// TIA Portal V17 export
// export: Created 2025-06-20T11:06:35.1143958Z, ExportSetting WithDefaults, DisplayName Totally Integrated Automation Portal, DisplayVersion V17 Update 8, DisplayName TIA Portal Openness, DisplayVersion V17 Update 8, DisplayName TIA Portal Version Control Interface, DisplayVersion V17, DisplayName SINAMICS Startdrive Advanced, DisplayVersion V17 SP2, DisplayName SINAMICS Startdrive G110M, G120, G120C, G120D, G120P, G115D, DisplayVersion V17 SP2, DisplayName SINAMICS Startdrive G130, G150, S120, S150, SINAMICS MV, S210, DisplayVersion V17 SP2, DisplayName STEP 7 Professional, DisplayVersion V17 Update 8, DisplayName SINUMERIK ONE STEP 7 Toolbox, DisplayVersion V17 Update 12, DisplayName SINUMERIK ONE PLC Basic Program Plus, DisplayVersion V17 Update 12, DisplayName SINUMERIK 840D sl STEP 7 Toolbox, DisplayVersion V17 Update 12, DisplayName STEP 7 Safety, DisplayVersion V17 Update 6, DisplayName WinCC Advanced, DisplayVersion V17 Update 8
DATA_BLOCK "DB1251_PART_CYCLE_UNIT_2"   // DB1251
{ S7_Optimized_Access := 'FALSE'; DB_Accessible_From_OPC_UA := 'FALSE' }
AUTHOR : ETXETAR
VERSION : 1.0
// stored: AutoNumber false, DBAccessibleFromOPCUA false, DBAccessibleFromWebserver true, IsOnlyStoredInLoadMemory false, IsWriteProtectedInAS false
   VAR RETAIN
      SEQUENCE : "SEQUENCE";
      CYCLE_UNIT_02_STATION_0 : Bool;   // CYCLE UNIT 02 STATION 0 START REQUEST
      CYCLE_UNIT_02_STATION_1 : Bool;   // CYCLE UNIT 02 STATION 1 START REQUEST
      CYCLE_UNIT_02_STATION_2 : Bool;   // CYCLE UNIT 02 STATION 2 START REQUEST
      CYCLE_UNIT_02_STATION_3 : Bool;   // CYCLE UNIT 02 STATION 3 START REQUEST
      CYCLE_UNIT_02_STATION_4 : Bool;   // CYCLE UNIT 02 STATION 4 START REQUEST
      UNIT_02_CALIBRATION_STATION_2 : Bool;   // UNIT 02 STATION 2 CALIBRATION CYCLE REQUEST
      UNIT_02_CALIBRATION_STATION_3 : Bool;   // UNIT 02 STATION 3 CALIBRATION CYCLE REQUEST
      UNIT_02_MASTER_MEASUREMENT_STATION_2 : Bool;   // UNIT 02 STATION 2 MASTER MEASUREMENT CYCLE REQUEST
      UNIT_02_MASTER_MEASUREMENT_STATION_3 : Bool;   // UNIT 02 STATION 3 MASTER MEASUREMENT CYCLE REQUEST
      U02_STA_1_COND_OK_STA_0_CYCLE : Bool;   // UNIT 02 STATION 1 CONDITIONS OK FOR STATION 0 CYCLE REQUEST
      U02_STA_2_COND_OK_STA_0_CYCLE : Bool;   // UNIT 02 STATION 2 CONDITIONS OK FOR STATION 0 CYCLE REQUEST
      U02_STA_3_COND_OK_STA_0_CYCLE : Bool;   // UNIT 02 STATION 3 CONDITIONS OK FOR STATION 0 CYCLE REQUEST
      U02_STA_4_COND_OK_STA_0_CYCLE : Bool;   // UNIT 02 STATION 4 CONDITIONS OK FOR STATION 0 CYCLE REQUEST
      U02_NEW_FACE_STA_1 : Bool;   // UNIT 02 NEW FACE IN STATION 1
      U02_FACE_DONE_STA_1 : Bool;   // UNIT 02 FACE DONE IN STATION 1
      FULL_DEPTH : Bool;   // FULL DEPTH
   END_VAR
BEGIN
   SEQUENCE.TIMER_TIME_EXCEED.PT := T#13M20S;
END_DATA_BLOCK
